FUNCTION_BLOCK FB_Kuka_KRC4 EXTENDS FB_Robot
VAR_INPUT
    HardwareInputs : st_Robot_Input;
END_VAR
VAR_OUTPUT
    HardwareOutputs : st_Robot_Output;
END_VAR
VAR    
    StartupTimeoutTON : TON := (PT:=T#7S);
END_VAR



ExecuteState();
IF NOT (nextState = curState) THEN
	StateTransition();
END_IF;

ACTION ExecuteState:
// Watch for safety inputs from robot, e-stops, etc. and immediately goto state error
// IF RobotSafetyInput THEN
//  curState := eState_Error;
// END_IF


CASE curState OF
	eState_Idle: ExecuteState_Idle();
	eState_Startup: ExecuteState_Startup();
	eState_Running: ExecuteState_Running();
	eState_Complete: ExecuteState_Complete();
	eState_Error: ExecuteState_Error();
	eState_Independent: ExecuteState_Independent();
END_CASE
END_ACTION

ACTION ExecuteState_Complete:
//Output signals

nextState := eState_Idle;
END_ACTION

ACTION ExecuteState_Error:
//Output signals
HardwareOutputs.fault := TRUE;
END_ACTION

ACTION ExecuteState_Held:
//Set outputs
END_ACTION

ACTION ExecuteState_Holding:
//Set outputs

//Wait for held signal, then go to Held state
nextState := eState_Held;
END_ACTION

ACTION ExecuteState_Idle:
// monitor IO while idle
// set IO while in idle state

//Output signals
HardwareOutputs.fault := FALSE;
END_ACTION

ACTION ExecuteState_Independent:
//Output signals
END_ACTION

ACTION ExecuteState_Running:
//Output signals
END_ACTION

ACTION ExecuteState_Startup:
nextState := eState_Running;
END_ACTION

METHOD hold : BOOL
IF curState = eState_Running THEN
	nextState := eState_Holding;
	hold := TRUE;
ELSE
	hold := FALSE;
END_IF
END_METHOD

METHOD reset : BOOL
resetAlarms();

IF curState = eState_Complete THEN
	nextState := eState_Idle;
	reset := TRUE;
ELSIF curState = eState_Error THEN
	nextState := eState_Idle;
	reset := TRUE;
ELSE
	reset := FALSE;
END_IF
END_METHOD

METHOD start: BOOL
VAR_INPUT
END_VAR
IF curState = eState_Idle THEN
	nextState := eState_Startup;
	start := TRUE;
ELSE
	start := FALSE;
END_IF
END_METHOD

ACTION StateTransition:
//reset timers watchdog timers

SUPER^.StateTransition();
END_ACTION

END_FUNCTION_BLOCK

(* stored: Version 1.1.0.1, ProductVersion 3.1.4024.9
   POU FB_Kuka_KRC4: Id {f8d86418-cb86-4d45-8e78-555e2b732be9}, SpecialFunc None
   Folder StateMachine: Id {7c66d7e1-2488-4916-8e34-5415c7b728b8}
   Folder States: Id {7937b9fc-d23c-4ba8-8e4c-d71968fa351b}
   Action ExecuteState: Id {b952fd7b-3836-4c2a-9f58-512de66cf7ba}
   Action ExecuteState_Complete: Id {2741ec13-6e13-409c-b94d-f6839e371abb}
   Action ExecuteState_Error: Id {980fe57f-81de-4517-9af8-7133844f06e0}
   Action ExecuteState_Held: Id {5c628b4c-c5ce-4679-a0f8-ae78f654952a}
   Action ExecuteState_Holding: Id {e231daa3-86b0-4899-94e0-9701642c16f3}
   Action ExecuteState_Idle: Id {a2798b24-d76f-4ec0-95b5-e6b9e123a8a4}
   Action ExecuteState_Independent: Id {b65891de-2ea1-4805-88bc-30b0afbbfb45}
   Action ExecuteState_Running: Id {a5ba05e4-9400-4de7-9da9-e7a4b1af2b4f}
   Action ExecuteState_Startup: Id {e404ca6a-06b8-4647-96a1-0eba31611d99}
   Method hold: Id {891f096c-804c-434c-a712-7f0e03019d21}
   Method reset: Id {f19f2312-87fc-4eb2-b020-267bf4ec89b1}
   Method start: Id {d39caee6-a1bc-408f-b1bc-380d00b162d4}
   Action StateTransition: Id {f5542f9f-b406-4151-94ab-c64519401327} *)
